INTERFACE IPage EXTENDS IObject, CNM_AoC.IHaveValue

METHOD addSuccessor
VAR_INPUT
	successor :CNM_AoC.IHaveValue;
END_VAR
END_METHOD

END_INTERFACE

(* stored: Version 1.1.0.1
   Itf IPage: Id {75a07323-c861-4cd5-a1b7-09f4c3448491}
   Method addSuccessor: Id {4e32ad3d-36da-4070-9f77-dae4a2af665b} *)
